VAR_GLOBAL
	
END_VAR

(* stored: Version 1.1.0.1, ProductVersion 3.1.4018.2
   GVL GVL_Status: Id {3bc995fb-5a01-423a-8a57-7019a9fd5bac} *)
